FUNCTION_BLOCK FB_StringBuilderEnumerator EXTENDS FB_AbstractStringEnumerator
VAR
	_ipStringBuilder : I_StringBuilder; 
END_VAR

(* Gets current string element*)
PROPERTY Current : T_LongString
GET
IF THIS^._ipStringBuilder = 0 THEN RETURN; END_IF
Current := THIS^._ipStringBuilder.GetChar(THIS^._Index);
END_GET
END_PROPERTY

(* !!!UNSAFE!!! DON'T FORGET TO RELEASE/DELETE FROM	MEMORY WHEN DONE!
 | Get a copy of the current element as a string buffer whose size is string length + 1.*)
METHOD Current_Buffer
VAR_IN_OUT
	pBuffer	: POINTER TO BYTE;
END_VAR
VAR
	pTemp : POINTER TO STRING;
END_VAR
IF THIS^._ipStringBuilder = 0 OR THIS^._Index < 0 OR_ELSE THIS^._Index >= THIS^._ipStringBuilder.Length THEN RETURN; END_IF
pTemp := __NEW(BYTE, 2);
pTemp^ := THIS^._ipStringBuilder.GetChar(THIS^._Index);
END_METHOD

{attribute 'hide'}
METHOD FB_init : BOOL
VAR_INPUT
	bInitRetains : BOOL; // if TRUE, the retain variables are initialized (warm start / cold start)
	bInCopyCode : BOOL;  // if TRUE, the instance afterwards gets moved into the copy code (online change)
	ipStringBuilder : I_StringBuilder;
END_VAR
THIS^._ipStringBuilder := ipStringBuilder;
END_METHOD

(* Gets current element. Returns TRUE if retrieval and converstion was successful. *)
METHOD GetCurrent : BOOL
VAR_INPUT
	sValue : REFERENCE TO STRING;
END_VAR
IF THIS^._ipStringBuilder = 0 THEN RETURN; END_IF
sValue := THIS^._ipStringBuilder.GetChar(THIS^._Index);
GetCurrent := TRUE;
END_METHOD

(* Advances enumerator to the next element. On first call or after reset it generates new element data to enumerate over.*)
METHOD Next : BOOL
IF THIS^._ipStringBuilder = 0 OR_ELSE THIS^._Index >= THIS^._ipStringBuilder.Length THEN RETURN; END_IF
THIS^._Index := THIS^._Index + 1;
Next := TRUE;
END_METHOD

END_FUNCTION_BLOCK

(* stored: Version 1.1.0.1, ProductVersion 3.1.4024.4
   POU FB_StringBuilderEnumerator: Id {8466a430-5af8-4804-a6cb-921d1b446bf2}, SpecialFunc None
   Property Current: Id {1c7c360b-0e9b-4fd3-ae58-c1c887921a7a}
   Get Get: Id {4a928de9-691d-4c6d-a864-501d08540cb0}
   Method Current_Buffer: Id {4904974d-69e1-4228-b332-9562133506ec}
   Method FB_init: Id {21e682db-2486-4e1a-8336-3adf2ff969ac}
   Method GetCurrent: Id {81506a7b-b59e-4636-9497-1499fe73fcf4}
   Method Next: Id {a591dc31-20cc-4208-83ed-070042ee01f5} *)
